Universal Robots PolyScope program: AlvarezZavaleta-LuisAlberto-P3.urp

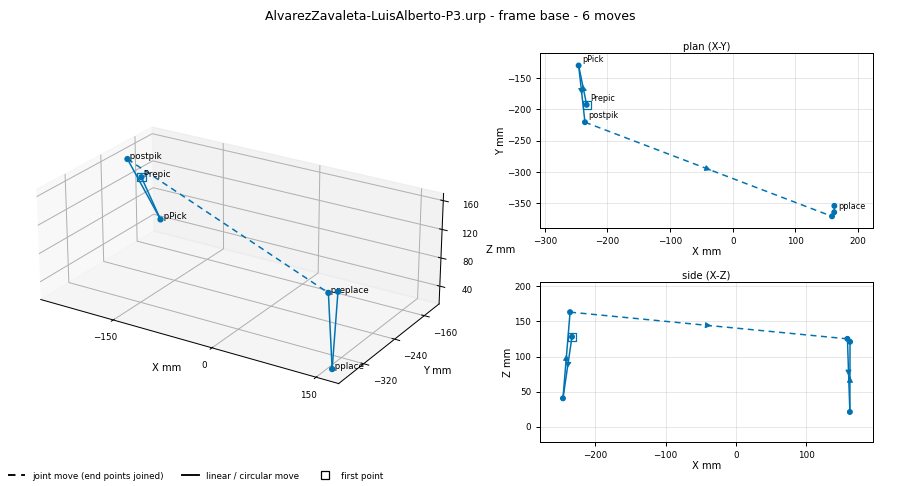
[picture p0: tool path of AlvarezZavaleta-LuisAlberto-P3.urp in frame base, 6 of 8 moves have a stored position in this frame; points joined in program order, loops and branches not executed]
Program AlvarezZavaleta-LuisAlberto-P3 (installation=default directory=/home/ur/ursim-current/programs createdIn=5.14.5 lastSavedIn=5.14.5 robotSerialNumber=20195399999)
Calibrated DH parameters: a=[0, -0.24355, -0.2132, 0, 0, 0]; d=[0.15185, 0, 0, 0.13105, 0.08535, 0.0921]; alpha=[1.570796, 0, 0, 1.570796, -1.570796, 0]; deltaTheta=[0, 0, 0, 0, 0, 0]
InitVariablesNode
BeforeStart
  P_ini := get_actual_tcp_pose()
  Alt_ini := P_ini[2]
  If Alt_ini<0.1
    Alt_ini := 0.12
    Script: P_ini[2] = Alt_ini
  MoveL speed 250 mm/s, acceleration 1200 mm/s^2 (useActiveTCP=true) feature=Base
    Waypoint Variable (Variable): variable=P_ini
  Wait Sleep waitTime=0.5
Robot Program (runOnlyOnce=true)
  MoveJ speed 80 deg/s, acceleration 120 deg/s^2 (useActiveTCP=true) feature=Base
    SuppressedNode
      deplazamiento := p[-150/1000,0,0,0,0,0]
    SuppressedNode
      Pre_pick := pose_add(P_ini, deplazamiento)
    Waypoint Prepic: motionParameters(blendRadius=0.05); TCP in base x=-233.193 y=-192.673 z=128.149 mm, rx=0.6007 ry=0.2378 rz=-0.5124 rad; joints [-105.365, -99.196, -81.485, -100.981, 83.413, -555.584] deg; TCP offset x=-0.83 y=-37.401 z=169.485 mm, rx=-2.6523 ry=-0.7245 rz=-0.1537 rad
  MoveL speed 300 mm/s, acceleration 1500 mm/s^2 (useActiveTCP=true) feature=Base
    SuppressedNode
      deplazamiento := p[0,0,-100/1000,0,0,0]
    SuppressedNode
      P_pick := pose_add(Pre_pick, deplazamiento)
    Waypoint pPick: TCP in base x=-246.017 y=-129.901 z=40.626 mm, rx=0.6011 ry=0.2377 rz=-0.5124 rad; joints [-111.229, -94.166, -111.848, -74.928, 82.273, -561.164] deg
    Wait Sleep waitTime=0.25
    Set DigitalOutput pin=digital_out[5]; digitalValue=1
    Wait Sleep waitTime=0.25
  MoveL speed 125 mm/s, acceleration 600 mm/s^2 (useActiveTCP=true) feature=Base
    SuppressedNode
      deplazamiento := p[0,0,150/1000,0,0,0]
    SuppressedNode
      Post_pick := pose_add(P_pick, deplazamiento)
    Waypoint postpik: motionParameters(blendRadius=0.05); TCP in base x=-235.912 y=-220.432 z=163.209 mm, rx=0.6012 ry=0.2378 rz=-0.5125 rad; joints [-104.604, -106.392, -62.952, -112.427, 83.534, -554.911] deg
  MoveJ speed 45 deg/s, acceleration 60 deg/s^2 (useActiveTCP=true) feature=Base
    Waypoint preplace: motionParameters(blendRadius=0.05); TCP in base x=158.615 y=-370.755 z=125.244 mm, rx=0.0663 ry=-0.0258 rz=-0.2406 rad; joints [-45.886, -97.394, -93.357, -59.685, 83.946, -512.913] deg; TCP offset x=-0.83 y=-37.401 z=169.485 mm, rx=-2.6523 ry=-0.7245 rz=-0.1537 rad
    SuppressedNode
      deplazamiento := p[300/1000,0,0,0,0,0]
    SuppressedNode
      Pre_place := pose_add(Post_pick, deplazamiento)
  MoveL speed 200 mm/s, acceleration 600 mm/s^2 (useActiveTCP=true) feature=Base
    SuppressedNode
      deplazamiento := p[0,0,-150/1000,0,0,0]
    SuppressedNode
      P_place := pose_add(Pre_place, deplazamiento)
    Waypoint pplace: TCP in base x=162.104 y=-364.22 z=21.199 mm, rx=0.0663 ry=-0.0258 rz=-0.2406 rad; joints [-44.664, -106.773, -112.527, -31.298, 83.408, -511.554] deg; TCP offset x=-0.83 y=-37.401 z=169.485 mm, rx=-2.6523 ry=-0.7245 rz=-0.1537 rad
    Wait Sleep waitTime=0.25
    Set DigitalOutput pin=digital_out[5]; digitalValue=0
    Wait Sleep waitTime=0.25
  MoveL speed 300 mm/s, acceleration 1500 mm/s^2 (useActiveTCP=true) feature=Base
    SuppressedNode
      deplazamiento := p[0,0,100/1000,0,0,0]
    SuppressedNode
      Post_place := pose_add(P_place, deplazamiento)
    Waypoint postplace: motionParameters(blendRadius=0.05); TCP in base x=162.338 y=-354.016 z=121.067 mm, rx=0.1299 ry=-0.0181 rz=-0.2414 rad; joints [-45.385, -97.32, -92.814, -63.03, 86.232, -511.66] deg
  MoveJ speed 80 deg/s, acceleration 120 deg/s^2 (useActiveTCP=true) feature=Base
    Waypoint Variable (Variable): variable=P_ini
